(SA := 16#21, SPN_Dest := 16578, Fmi_Dest := 31, FmiExt_Dest := 255, SPN_Src := 16578, Fmi_Src := 31, Assembly := 255, CompType := 255, CompFunc := 255, Symbol := "", AccLevel := 16#AAAA, ErrorType := eErrorType.ERROR, ErrorSeverity := eErrorSeverity.CAT5_MALFUNCTION, ErrorDescriptionIndex := _eDm1ErrorText.txt_Err_Spn16578_Fmi31_FmiExt255), (SA := 16#20, SPN_Dest := 16583, Fmi_Dest := 31, FmiExt_Dest := 255, SPN_Src := 16583, Fmi_Src := 31, Assembly := 255, CompType := 255, CompFunc := 255, Symbol := "", AccLevel := 16#AAAA, ErrorType := eErrorType.ERROR, ErrorSeverity := eErrorSeverity.CAT5_MALFUNCTION, ErrorDescriptionIndex := _eDm1ErrorText.txt_Err_Spn16583_Fmi31_FmiExt255), (SA := 16#21, SPN_Dest := 16588, Fmi_Dest := 31, FmiExt_Dest := 255, SPN_Src := 16588, Fmi_Src := 31, Assembly := 255, CompType := 255, CompFunc := 255, Symbol := "", AccLevel := 16#AAAA, ErrorType := eErrorType.ERROR, ErrorSeverity := eErrorSeverity.CAT5_MALFUNCTION, ErrorDescriptionIndex := _eDm1ErrorText.txt_Err_Spn16588_Fmi31_FmiExt255), (SA := 16#21, SPN_Dest := 16589, Fmi_Dest := 31, FmiExt_Dest := 255, SPN_Src := 16589, Fmi_Src := 31, Assembly := 255, CompType := 255, CompFunc := 255, Symbol := "", AccLevel := 16#AAAA, ErrorType := eErrorType.ERROR, ErrorSeverity := eErrorSeverity.CAT5_MALFUNCTION, ErrorDescriptionIndex := _eDm1ErrorText.txt_Err_Spn16589_Fmi31_FmiExt255), (SA := 16#21, SPN_Dest := 16590, Fmi_Dest := 31, FmiExt_Dest := 255, SPN_Src := 16590, Fmi_Src := 31, Assembly := 255, CompType := 255, CompFunc := 255, Symbol := "", AccLevel := 16#AAAA, ErrorType := eErrorType.ERROR, ErrorSeverity := eErrorSeverity.CAT0_NO, ErrorDescriptionIndex := _eDm1ErrorText.txt_Err_Spn16590_Fmi31_FmiExt255), (SA := 16#21, SPN_Dest := 16591, Fmi_Dest := 31, FmiExt_Dest := 255, SPN_Src := 16591, Fmi_Src := 31, Assembly := 255, CompType := 255, CompFunc := 255, Symbol := "", AccLevel := 16#AAAA, ErrorType := eErrorType.ERROR, ErrorSeverity := eErrorSeverity.CAT0_NO, ErrorDescriptionIndex := _eDm1ErrorText.txt_Err_Spn16591_Fmi31_FmiExt255), (SA := 16#21, SPN_Dest := 16592, Fmi_Dest := 31, FmiExt_Dest := 255, SPN_Src := 16592, Fmi_Src := 31, Assembly := 255, CompType := 255, CompFunc := 255, Symbol := "", AccLevel := 16#AAAA, ErrorType := eErrorType.ERROR, ErrorSeverity := eErrorSeverity.CAT0_NO, ErrorDescriptionIndex := _eDm1ErrorText.txt_Err_Spn16592_Fmi31_FmiExt255), (SA := 16#21, SPN_Dest := 16593, Fmi_Dest := 31, FmiExt_Dest := 255, SPN_Src := 16593, Fmi_Src := 31, Assembly := 255, CompType := 255, CompFunc := 255, Symbol := "", AccLevel := 16#AAAA, ErrorType := eErrorType.ERROR, ErrorSeverity := eErrorSeverity.CAT0_NO, ErrorDescriptionIndex := _eDm1ErrorText.txt_Err_Spn16593_Fmi31_FmiExt255), (SA := 16#21, SPN_Dest := 16595, Fmi_Dest := 31, FmiExt_Dest := 255, SPN_Src := 16595, Fmi_Src := 31, Assembly := 255, CompType := 255, CompFunc := 255, Symbol := "", AccLevel := 16#AAAA, ErrorType := eErrorType.ERROR, ErrorSeverity := eErrorSeverity.CAT5_MALFUNCTION, ErrorDescriptionIndex := _eDm1ErrorText.txt_Err_Spn16595_Fmi31_FmiExt255), (SA := 16#21, SPN_Dest := 16596, Fmi_Dest := 31, FmiExt_Dest := 255, SPN_Src := 16596, Fmi_Src := 31, Assembly := 255, CompType := 255, CompFunc := 255, Symbol := "", AccLevel := 16#AAAA, ErrorType := eErrorType.ERROR, ErrorSeverity := eErrorSeverity.CAT0_NO, ErrorDescriptionIndex := _eDm1ErrorText.txt_Err_Spn16596_Fmi31_FmiExt255), (SA := 16#21, SPN_Dest := 16597, Fmi_Dest := 31, FmiExt_Dest := 255, SPN_Src := 16597, Fmi_Src := 31, Assembly := 255, CompType := 255, CompFunc := 255, Symbol := "", AccLevel := 16#AAAA, ErrorType := eErrorType.ERROR, ErrorSeverity := eErrorSeverity.CAT0_NO, ErrorDescriptionIndex := _eDm1ErrorText.txt_Err_Spn16597_Fmi31_FmiExt255), (SA := 16#21, SPN_Dest := 16598, Fmi_Dest := 31, FmiExt_Dest := 255, SPN_Src := 16598, Fmi_Src := 31, Assembly := 255, CompType := 255, CompFunc := 255, Symbol := "", AccLevel := 16#AAAA, ErrorType := eErrorType.ERROR, ErrorSeverity := eErrorSeverity.CAT0_NO, ErrorDescriptionIndex := _eDm1ErrorText.txt_Err_Spn16598_Fmi31_FmiExt255), (SA := 16#21, SPN_Dest := 16599, Fmi_Dest := 31, FmiExt_Dest := 255, SPN_Src := 16599, Fmi_Src := 31, Assembly := 255, CompType := 255, CompFunc := 255, Symbol := "", AccLevel := 16#AAAA, ErrorType := eErrorType.ERROR, ErrorSeverity := eErrorSeverity.CAT0_NO, ErrorDescriptionIndex := _eDm1ErrorText.txt_Err_Spn16599_Fmi31_FmiExt255), (SA := 16#21, SPN_Dest := 16611, Fmi_Dest := 31, FmiExt_Dest := 255, SPN_Src := 16611, Fmi_Src := 31, Assembly := 255, CompType := 255, CompFunc := 255, Symbol := "", AccLevel := 16#AAAA, ErrorType := eErrorType.ERROR, ErrorSeverity := eErrorSeverity.CAT5_MALFUNCTION, ErrorDescriptionIndex := _eDm1ErrorText.txt_Err_Spn16611_Fmi31_FmiExt255), (SA := 16#21, SPN_Dest := 16612, Fmi_Dest := 31, FmiExt_Dest := 255, SPN_Src := 16612, Fmi_Src := 31, Assembly := 255, CompType := 255, CompFunc := 255, Symbol := "", AccLevel := 16#AAAA, ErrorType := eErrorType.ERROR, ErrorSeverity := eErrorSeverity.CAT5_MALFUNCTION, ErrorDescriptionIndex := _eDm1ErrorText.txt_Err_Spn16612_Fmi31_FmiExt255), (SA := 16#21, SPN_Dest := 16613, Fmi_Dest := 31, FmiExt_Dest := 255, SPN_Src := 16613, Fmi_Src := 31, Assembly := 255, CompType := 255, CompFunc := 255, Symbol := "", AccLevel := 16#AAAA, ErrorType := eErrorType.ERROR, ErrorSeverity := eErrorSeverity.CAT5_MALFUNCTION, ErrorDescriptionIndex := _eDm1ErrorText.txt_Err_Spn16613_Fmi31_FmiExt255), (SA := 16#21, SPN_Dest := 16614, Fmi_Dest := 31, FmiExt_Dest := 255, SPN_Src := 16614, Fmi_Src := 31, Assembly := 255, CompType := 255, CompFunc := 255, Symbol := "", AccLevel := 16#AAAA, ErrorType := eErrorType.ERROR, ErrorSeverity := eErrorSeverity.CAT5_MALFUNCTION, ErrorDescriptionIndex := _eDm1ErrorText.txt_Err_Spn16614_Fmi31_FmiExt255)];
  DM1_SPN_SRC_MIN_New_Master_List : UDINT := 1000;
  DM1_SPN_MAX_New_Master_List : UDINT := 16614;
END_VAR

VAR_GLOBAL CONSTANT  (* DM1ErrorGroups *)
  GroupCount : INT := 3;
  g_ErrorCategoryGroups : ARRAY[0..(GroupCount - 1)] OF TErrorGroup := [(ErrorType := eErrorType.INFO, Behaviour := [(ErrorSeverity := eErrorSeverity.CAT0_NO, AcousticWarningOnActivation := eSwitchState.OFF, AcousticWarningUntilConfirmation := eBeepSignal.OFF, AcousticWarningAfterConfirmation := eBeepSignal.OFF, ShowOnIgnition := eSwitchState.ON, ShowPopup := 0), (ErrorSeverity := eErrorSeverity.CAT1_WHITE, AcousticWarningOnActivation := eSwitchState.OFF, AcousticWarningUntilConfirmation := eBeepSignal.OFF, AcousticWarningAfterConfirmation := eBeepSignal.OFF, ShowOnIgnition := eSwitchState.ON, ShowPopup := 0), (ErrorSeverity := eErrorSeverity.CAT2_YELLOW, AcousticWarningOnActivation := eSwitchState.ON, AcousticWarningUntilConfirmation := eBeepSignal.OFF, AcousticWarningAfterConfirmation := eBeepSignal.OFF, ShowOnIgnition := eSwitchState.OFF, ShowPopup := 0), (ErrorSeverity := eErrorSeverity.CAT3_AMBER, AcousticWarningOnActivation := eSwitchState.ON, AcousticWarningUntilConfirmation := eBeepSignal.SLOW, AcousticWarningAfterConfirmation := eBeepSignal.OFF, ShowOnIgnition := eSwitchState.OFF, ShowPopup := 0), (ErrorSeverity := eErrorSeverity.CAT4_RED, AcousticWarningOnActivation := eSwitchState.ON, AcousticWarningUntilConfirmation := eBeepSignal.SLOW, AcousticWarningAfterConfirmation := eBeepSignal.SLOW, ShowOnIgnition := eSwitchState.OFF, ShowPopup := 0), (ErrorSeverity := eErrorSeverity.CAT5_MALFUNCTION, AcousticWarningOnActivation := eSwitchState.ON, AcousticWarningUntilConfirmation := eBeepSignal.PERMANENT, AcousticWarningAfterConfirmation := eBeepSignal.PERMANENT, ShowOnIgnition := eSwitchState.OFF, ShowPopup := 0)]), (ErrorType := eErrorType.WARNING, Behaviour := [(ErrorSeverity := eErrorSeverity.CAT0_NO, AcousticWarningOnActivation := eSwitchState.OFF, AcousticWarningUntilConfirmation := eBeepSignal.OFF, AcousticWarningAfterConfirmation := eBeepSignal.OFF, ShowOnIgnition := eSwitchState.ON, ShowPopup := 0), (ErrorSeverity := eErrorSeverity.CAT1_WHITE, AcousticWarningOnActivation := eSwitchState.OFF, AcousticWarningUntilConfirmation := eBeepSignal.OFF, AcousticWarningAfterConfirmation := eBeepSignal.OFF, ShowOnIgnition := eSwitchState.ON, ShowPopup := 0), (ErrorSeverity := eErrorSeverity.CAT2_YELLOW, AcousticWarningOnActivation := eSwitchState.ON, AcousticWarningUntilConfirmation := eBeepSignal.OFF, AcousticWarningAfterConfirmation := eBeepSignal.OFF, ShowOnIgnition := eSwitchState.OFF, ShowPopup := 0), (ErrorSeverity := eErrorSeverity.CAT3_AMBER, AcousticWarningOnActivation := eSwitchState.ON, AcousticWarningUntilConfirmation := eBeepSignal.SLOW, AcousticWarningAfterConfirmation := eBeepSignal.OFF, ShowOnIgnition := eSwitchState.OFF, ShowPopup := 0), (ErrorSeverity := eErrorSeverity.CAT4_RED, AcousticWarningOnActivation := eSwitchState.ON, AcousticWarningUntilConfirmation := eBeepSignal.SLOW, AcousticWarningAfterConfirmation := eBeepSignal.SLOW, ShowOnIgnition := eSwitchState.OFF, ShowPopup := 0), (ErrorSeverity := eErrorSeverity.CAT5_MALFUNCTION, AcousticWarningOnActivation := eSwitchState.ON, AcousticWarningUntilConfirmation := eBeepSignal.PERMANENT, AcousticWarningAfterConfirmation := eBeepSignal.PERMANENT, ShowOnIgnition := eSwitchState.OFF, ShowPopup := 0)]), (ErrorType := eErrorType.ERROR, Behaviour := [(ErrorSeverity := eErrorSeverity.CAT0_NO, AcousticWarningOnActivation := eSwitchState.OFF, AcousticWarningUntilConfirmation := eBeepSignal.OFF, AcousticWarningAfterConfirmation := eBeepSignal.OFF, ShowOnIgnition := eSwitchState.ON, ShowPopup := 0), (ErrorSeverity := eErrorSeverity.CAT1_WHITE, AcousticWarningOnActivation := eSwitchState.OFF, AcousticWarningUntilConfirmation := eBeepSignal.OFF, AcousticWarningAfterConfirmation := eBeepSignal.OFF, ShowOnIgnition := eSwitchState.ON, ShowPopup := 0), (ErrorSeverity := eErrorSeverity.CAT2_YELLOW, AcousticWarningOnActivation := eSwitchState.ON, AcousticWarningUntilConfirmation := eBeepSignal.OFF, AcousticWarningAfterConfirmation := eBeepSignal.OFF, ShowOnIgnition := eSwitchState.OFF, ShowPopup := 0), (ErrorSeverity := eErrorSeverity.CAT3_AMBER, AcousticWarningOnActivation := eSwitchState.ON, AcousticWarningUntilConfirmation := eBeepSignal.OFF, AcousticWarningAfterConfirmation := eBeepSignal.OFF, ShowOnIgnition := eSwitchState.OFF, ShowPopup := -1), (ErrorSeverity := eErrorSeverity.CAT4_RED, AcousticWarningOnActivation := eSwitchState.ON, AcousticWarningUntilConfirmation := eBeepSignal.OFF, AcousticWarningAfterConfirmation := eBeepSignal.OFF, ShowOnIgnition := eSwitchState.OFF, ShowPopup := -1), (ErrorSeverity := eErrorSeverity.CAT5_MALFUNCTION, AcousticWarningOnActivation := eSwitchState.ON, AcousticWarningUntilConfirmation := eBeepSignal.OFF, AcousticWarningAfterConfirmation := eBeepSignal.OFF, ShowOnIgnition := eSwitchState.OFF, ShowPopup := -1)])];
END_VAR

FUNCTION MatchLibInit_DM1 : BOOL

            // **********************************************************************************************************************
// *  AUTO-GENERATED:  PdtCodeBuilder.dll (Version: 1.2.7, Build: 080)
// *  Itf-Version:     1.7.0
// *  Pdt-Version:     2.11.72.172
// *  Pdt-ProjVersion: 0.0.0
// *  Match-Version:   07.04.00.00
// *  Copyright (C) 2012 HYDAC SYSTEM GMBH -  All rights reserved.
// *  Entwicklungsbüro Berlin - Zum Kiesberg 16 - D-14979 Großbeeren
// *  2025-04-18 16:40:50 created
// **********************************************************************************************************************
gLib_MatchInitializer.Dm1[0].LanguageCount := DM1_LANGUAGE_COUNT;
gLib_MatchInitializer.Dm1[0].FMICount := DM1_FMI_COUNT;
gLib_MatchInitializer.Dm1[0].FMIEXCount := DM1_FMIEX_COUNT;
gLib_MatchInitializer.Dm1[0].AssemblyCount := DM1_ASSEMBLY_COUNT;
gLib_MatchInitializer.Dm1[0].ComponentTypeCount := DM1_COMPONENTTYPE_COUNT;
gLib_MatchInitializer.Dm1[0].ComponentFunctionCount := DM1_COMPONENTFUNCTION_COUNT;

gLib_MatchInitializer.Dm1[0].NativeLanguageNames := ADR(g_DM1Texts_NativeLanguageName);
gLib_MatchInitializer.Dm1[0].FMITextsPointer := ADR(g_DM1Texts_FMI);
gLib_MatchInitializer.Dm1[0].FMIEXTextsPointer := ADR(g_DM1Texts_FMIEX);
gLib_MatchInitializer.Dm1[0].AssemblyTextsPointer := ADR(g_DM1Texts_Assembly);
gLib_MatchInitializer.Dm1[0].ComponentTypeTextsPointer := ADR(g_DM1Texts_ComponentType);
gLib_MatchInitializer.Dm1[0].ComponentFunctionTextsPointer := ADR(g_DM1Texts_ComponentFunction);

gLib_MatchInitializer.ErrorBehaviours := ADR(g_ErrorCategoryGroups);

gLib_MatchInitializer.Dm1[0].ErrorListEntries := DM1_SPN_SRC_COUNT_New_Master_List;
gLib_MatchInitializer.Dm1[0].ErrorListPointer := ADR(g_DM1_ErrorList_New_Master_List);
gLib_MatchInitializer.Dm1[0].SpnMin := DM1_SPN_SRC_MIN_New_Master_List;
gLib_MatchInitializer.Dm1[0].SpnMax := DM1_SPN_MAX_New_Master_List;

gLib_MatchInitializer.Dm1[0].DescriptionTextPointer := ADR(g_ErrTranslations);
gLib_MatchInitializer.Dm1[0].DescriptionCountPerLanguage := ERR_TRANSLATION_TEXT_COUNT;

          
END_FUNCTION
